{attribute addProperty BoxType "EL2252-0000-0016"}
{attribute addProperty Id "StartTimeAT %Q*ULINT648"}
{attribute addProperty CRC "3527759060"}
{attribute addProperty SizeInBites "64"}
{attribute addProperty SizeInBytes "8"}
TYPE DC_Sync_Start_D24554D4 :
STRUCT
	{attribute addProperty Name "StartTime"}
	StartTime AT %Q* : ULINT;
END_STRUCT
END_TYPE

(* stored: Version 1.2.0.0, ProductVersion 3.1.4024.9
   DUT DC_Sync_Start_D24554D4: Id {a1f4aa4b-90c0-402a-814a-1fd3beaa703b} *)
